// TIA Portal project "AvvioMacchinaIndustriale" (V20)

(* hardware
DEVICE "S7-1200 station_1"  S7-1200 Station
   slot 0: "Rack_0"  S7-1200 Rack  Rack  V1.0
   slot 1: "Playground_PLC"  CPU 1214C DC/DC/DC  6ES7 214-1AG40-0XB0  V4.7
   slot 3: "AQ 1x12BIT_1"  AQ1 signal board  6ES7 232-4HA30-0XB0  V1.0
*)

// ===== PLC "Playground_PLC"  CPU 1214C DC/DC/DC =====

VAR_GLOBAL   // PLC tag table "Default tag table"
   "KM1" AT %M0.0 : Bool;
   "P1" AT %M0.1 : Bool;
   "P2" AT %M0.2 : Bool;
   "P3" AT %M0.3 : Bool;
   "STOP" AT %M0.4 : Bool;
   "L" AT %M0.5 : Bool;
   "M1" AT %M0.6 : Bool;
   "M2" AT %M0.7 : Bool;
   "M3" AT %M1.0 : Bool;
   "HELPER_M1" AT %M1.1 : Bool;
   "HELPER_M2" AT %M1.2 : Bool;
   "HELPER_M3" AT %M1.3 : Bool;
END_VAR

ORGANIZATION_BLOCK "Main"   // OB1, LAD, ProgramCycle
TITLE = "Main Program Sweep (Cycle)"
{ S7_Optimized_Access := 'TRUE' }
VERSION : 0.1
   VAR_INPUT
      Initial_Call : Bool;   // Initial call of this OB
      Remanence : Bool;   // =True, if remanent data are available
   END_VAR
   VAR_TEMP   // added for the SCL form of the ladder/FBD networks
      _w1 : Bool;
      _w2 : Bool;
      _w3 : Bool;
   END_VAR
BEGIN

REGION Network 1
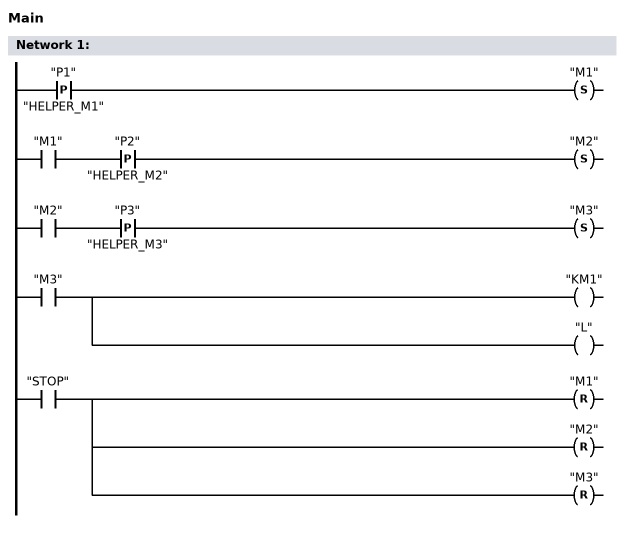
   RUNG wire#powerrail
      P_Contact(operand := "P1", bit := "HELPER_M1")
      S_Coil( "M1" )
   END_RUNG
   RUNG wire#powerrail
      Contact( "M1" )
      P_Contact(operand := "P2", bit := "HELPER_M2")
      S_Coil( "M2" )
   END_RUNG
   RUNG wire#powerrail
      Contact( "M2" )
      P_Contact(operand := "P3", bit := "HELPER_M3")
      S_Coil( "M3" )
   END_RUNG
   RUNG wire#powerrail
      Contact( "M3" )
      wire#w1
      Coil( "KM1" )
   END_RUNG
   RUNG wire#w1
      Coil( "L" )
   END_RUNG
   RUNG wire#powerrail
      Contact( "STOP" )
      wire#w2
      R_Coil( "M1" )
   END_RUNG
   RUNG wire#w2
      R_Coil( "M2" )
   END_RUNG
   RUNG wire#w2
      R_Coil( "M3" )
   END_RUNG
   // the same network as SCL:
   #_w1 := "P1" AND NOT "HELPER_M1";   // rising edge of "P1"
   "HELPER_M1" := "P1";
   IF #_w1 THEN "M1" := TRUE; END_IF;
   #_w2 := "M1" AND "P2" AND NOT "HELPER_M2";   // rising edge of "P2"
   "HELPER_M2" := "P2";
   IF #_w2 THEN "M2" := TRUE; END_IF;
   #_w3 := "M2" AND "P3" AND NOT "HELPER_M3";   // rising edge of "P3"
   "HELPER_M3" := "P3";
   IF #_w3 THEN "M3" := TRUE; END_IF;
   "KM1" := "M3";
   "L" := "M3";
   IF "STOP" THEN
       "M1" := FALSE;
       "M2" := FALSE;
       "M3" := FALSE;
   END_IF;
END_REGION
END_ORGANIZATION_BLOCK